Yaskawa INFORM job: A-1-08279-80-SUB-R.JBI

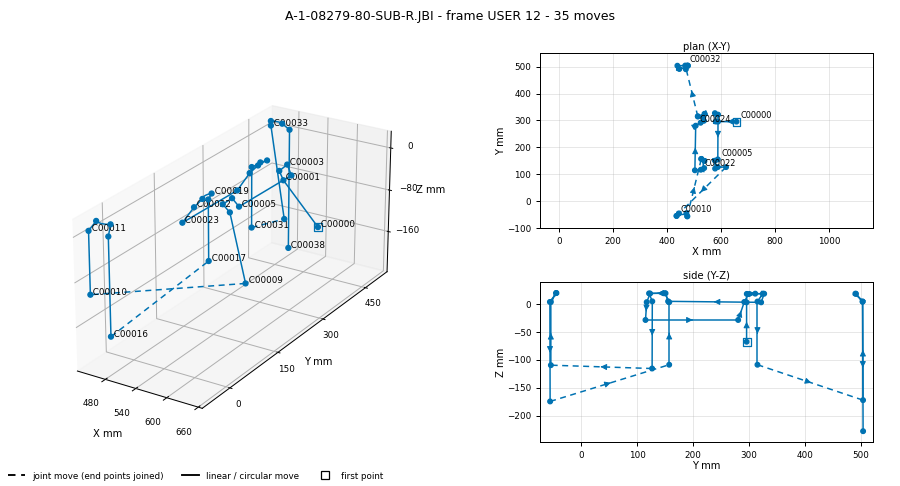
[picture p0: tool path of A-1-08279-80-SUB-R.JBI in frame USER 12, 35 of 39 moves have a stored position in this frame; points joined in program order, loops and branches not executed]
/JOB
//NAME A-1-08279-80-SUB-R
///FOLDERNAME PART_420-08279-80
//POS
///NPOS 39,0,39,0,0,0
///USER 12
///TOOL 4
///POSTYPE USER
///RECTAN
///RCONF 1,0,0,0,0,0,0,0,0,0,0,0,0,0,0,0,0,0,0,0,0,0,0,0
C00000=657.099,295.730,-67.432,-27.8961,11.3051,78.2351
C00001=588.519,295.721,3.021,-46.5250,6.9320,75.2540
C00002=579.969,296.078,18.126,-46.5258,6.9307,75.2543
C00003=577.041,327.152,18.437,-46.5237,6.9340,75.2552
C00004=588.755,321.720,3.021,-46.5250,6.9320,75.2540
C00005=587.773,155.478,4.815,-42.9430,-21.0870,89.6170
C00006=577.215,150.868,19.159,-42.9414,-21.0917,89.6143
C00007=577.842,121.423,19.065,-42.9383,-21.0890,89.6174
C00008=587.773,127.194,4.815,-42.9430,-21.0870,89.6170
C00009=618.287,126.871,-115.266,-42.9430,-21.0870,89.6170
C00010=434.578,-54.115,-109.298,-6.5594,-44.9787,-116.9695
C00011=434.802,-54.182,3.718,-6.5590,-44.9790,-116.9690
C00012=443.596,-44.809,19.622,-6.5595,-44.9791,-116.9648
C00013=455.754,-48.787,19.626,-6.5585,-44.9768,-90.5169
C00014=471.216,-44.177,19.737,-6.5552,-44.9816,-55.2600
C00015=474.608,-55.834,3.718,-6.5580,-44.9790,-55.2560
C00016=474.346,-55.448,-174.107,-6.5568,-44.9787,-55.2555
C00017=526.608,157.384,-108.500,-16.3490,-44.1220,152.7880
C00018=526.609,157.384,3.318,-16.3490,-44.1220,152.7880
C00019=538.213,149.581,19.290,-11.9916,-45.2337,146.5959
C00020=533.936,136.169,19.326,-16.5569,-44.9790,179.4784
C00021=537.166,123.301,18.778,-16.5155,-44.7739,-145.3158
C00022=524.621,117.175,3.331,-16.5140,-44.7720,-151.5720
C00023=502.748,115.031,-28.500,-16.5140,-44.7720,-151.5720
C00024=505.771,280.690,-28.500,3.4420,-44.9790,-154.0720
C00025=524.020,291.566,3.647,3.4420,-44.9790,-154.0720
C00026=536.186,298.815,17.769,3.4420,-44.9790,-154.0720
C00027=536.368,299.659,18.248,3.4082,-44.7464,-155.9617
C00028=533.310,311.158,18.544,7.8960,-43.2322,176.8585
C00029=538.425,324.844,18.609,15.6693,-44.9800,144.2140
C00030=513.589,315.156,4.472,16.5470,-44.9790,144.2150
C00031=513.589,315.156,-108.500,16.5470,-44.9790,144.2150
C00032=467.026,503.882,-171.799,28.9267,-36.2202,77.7079
C00033=437.809,503.258,4.353,28.9260,-36.2220,77.7090
C00034=445.033,491.127,18.426,28.9260,-36.2221,77.7084
C00035=456.382,494.214,18.496,15.7352,-42.8106,71.8260
C00036=469.182,490.167,18.479,13.1194,-43.5301,40.3815
C00037=476.884,503.018,4.353,12.3290,-43.7170,41.5290
C00038=476.283,503.967,-227.292,12.0360,-43.7828,41.9536
///TOOL 0
///POSTYPE ANGLE
///ANGLE
EC00000=-45.0000
///TOOL 4
EC00001=-45.0000
///TOOL 0
EC00002=-45.0000
EC00003=-45.0000
///TOOL 4
EC00004=-45.0000
EC00005=-45.0000
///TOOL 0
EC00006=-45.0005
EC00007=-45.0005
///TOOL 4
EC00008=-45.0000
EC00009=-45.0000
///TOOL 0
EC00010=-90.0000
///TOOL 4
EC00011=-90.0000
///TOOL 0
EC00012=-90.0000
EC00013=-90.0000
EC00014=-90.0000
///TOOL 4
EC00015=-90.0000
///TOOL 0
EC00016=-90.0000
///TOOL 4
EC00017=-90.0000
EC00018=-90.0000
///TOOL 0
EC00019=-90.0000
EC00020=-90.0000
EC00021=-90.0000
///TOOL 4
EC00022=-90.0000
EC00023=-90.0000
EC00024=-90.0000
EC00025=-90.0000
EC00026=-90.0000
///TOOL 0
EC00027=-90.0000
EC00028=-90.0000
EC00029=-90.0000
///TOOL 4
EC00030=-90.0000
EC00031=-90.0000
///TOOL 0
EC00032=-90.0000
///TOOL 4
EC00033=-90.0000
///TOOL 0
EC00034=-90.0000
EC00035=-90.0000
EC00036=-90.0000
///TOOL 4
EC00037=-90.0000
///TOOL 0
EC00038=-90.0000
//INST
///DATE 2021/10/29 11:36
///ATTR SC,RW,RJ
////FRAME USER 12
///GROUP1 RB1
///GROUP2 ST2
NOP
'Path Start: PP9
'Warning, the first motion progra
'mmed for this routine was not a
'joint motion
'The following movement has been
'added. Please update your OCTOPU
'Z simulation.
MOVJ C00000 VJ=100.00  +MOVJ EC00000
SMOVL C00001 V=1250.0  +MOVJ EC00001
SMOVL C00002 V=300.0  +MOVJ EC00002
ARCON ASF#(951)
SMOVL C00003 V=8.5  +MOVJ EC00003
ARCOF AEF#(951)
SMOVL C00004 V=1250.0  +MOVJ EC00004
'Path End
'Path Start: PP15
SMOVL C00005 V=1250.0  +MOVJ EC00005
SMOVL C00006 V=300.0  +MOVJ EC00006
ARCON ASF#(951)
SMOVL C00007  +MOVJ EC00007
ARCOF AEF#(951)
SMOVL C00008 V=1250.0  +MOVJ EC00008
SMOVL C00009 V=1250.0  +MOVJ EC00009
'Path End
'Path Start: PP16
MOVJ C00010 VJ=25.00  +MOVJ EC00010
SMOVL C00011 V=1250.0  +MOVJ EC00011
SMOVC C00012 V=300.0  +MOVJ EC00012
ARCON ASF#(951)
SMOVC C00013 V=8.5  +MOVJ EC00013
SMOVC C00014 V=8.5  +MOVJ EC00014
ARCOF AEF#(951)
SMOVL C00015 V=1250.0  +MOVJ EC00015
SMOVL C00016 V=1250.0  +MOVJ EC00016
'Path End
'Path Start: PP19
MOVJ C00017 VJ=100.00  +MOVJ EC00017
SMOVL C00018 V=1250.0  +MOVJ EC00018
SMOVC C00019 V=300.0  +MOVJ EC00019
ARCON ASF#(951)
SMOVC C00020 V=8.5  +MOVJ EC00020
SMOVC C00021 V=8.5  +MOVJ EC00021
ARCOF AEF#(951)
SMOVL C00022 V=1250.0  +MOVJ EC00022
SMOVL C00023 V=1250.0  +MOVJ EC00023
'Path End
'Path Start: PP20
SMOVL C00024 V=1250.0  +MOVJ EC00024
SMOVL C00025 V=1250.0  +MOVJ EC00025
SMOVC C00026 V=300.0  +MOVJ EC00026
ARCON ASF#(951)
SMOVC C00027 V=8.5  +MOVJ EC00027
SMOVC C00028 V=8.5  +MOVJ EC00028
SMOVC C00029 V=8.5  +MOVJ EC00029
ARCOF AEF#(951)
SMOVL C00030 V=1250.0  +MOVJ EC00030
SMOVL C00031 V=1250.0  +MOVJ EC00031
'Path End
'Path Start: PP22
MOVJ C00032 VJ=100.00  +MOVJ EC00032
SMOVL C00033 V=1250.0  +MOVJ EC00033
SMOVC C00034 V=300.0  +MOVJ EC00034
ARCON ASF#(951)
SMOVC C00035 V=8.5  +MOVJ EC00035
SMOVC C00036 V=8.5  +MOVJ EC00036
ARCOF AEF#(951)
SMOVL C00037 V=1250.0  +MOVJ EC00037
SMOVL C00038 V=1250.0  +MOVJ EC00038
'Path End
END
